// Struckig
// Copyright (C) 2022 Stefan Besler

// This program is free software: you can redistribute it and/or modify
// it under the terms of the GNU General Public License as published by
// the Free Software Foundation, either version 3 of the License, or
// (at your option) any later version.

// This program is distributed in the hope that it will be useful,
// but WITHOUT ANY WARRANTY; without even the implied warranty of
// MERCHANTABILITY or FITNESS FOR A PARTICULAR PURPOSE.  See the
// GNU General Public License for more details.
//
// You should have received a copy of the GNU General Public License
// along with THIS PROGRAM.  IF NOT, see <http://www.gnu.org/licenses/>.
/// Floating-point remainder operation.
/// Returns the remainder of `x / y` with truncation toward zero:
/// `x - TRUNC(x / y) * y`.
FUNCTION Fmod : LREAL
VAR_INPUT
  x : LREAL; //< Dividend.
  y : LREAL; //< Divisor.
END_VAR

Fmod := x - TRUNC(x / y) * y;

END_FUNCTION

(* stored: Version 1.1.0.1
   POU Fmod: Id {e7de841c-f3d1-4a5d-b60b-81609d8fb3bd}, SpecialFunc None *)
